(*
SPDX-FileCopyrightText: © 2026 Oleksandr Tiutyk <trofimich@gmail.com>
SPDX-License-Identifier: MIT
License: https://opensource.org/license/mit
*)

(*!
<summary>Provides lexical checks for directory and file path strings.</summary>
<description>
These checks perform no filesystem I/O, normalization or access checks. Passing does not certify acceptance by
a native service or target filesystem. The current filter is not a complete Windows, UNC or platform-specific
path validator; it does not validate reserved names or dot components. Callers must separately satisfy the
path requirements of the actual operation and target.
</description>
*)

{attribute 'no_explicit_call' := 'do not call this function block directly'}
PROGRAM PathHelper
VAR CONSTANT
	//! <summary>Drive-letter, colon and separator occupy the first three bytes of an absolute drive prefix.</summary>
	_DrivePrefixLength : UDINT := 3;
	//! <summary>Zero-based index of the colon immediately following a drive letter.</summary>
	_DriveColonIndex : UDINT := 1;
	//! <summary>Zero-based index of the separator following the drive colon.</summary>
	_DriveSeparatorIndex : UDINT := 2;
	//! <summary>Last index allowed in the initial separator pair before repeated separators are rejected.</summary>
	_LeadingSeparatorPairLastIndex : UDINT := 1;
END_VAR
VAR
	{attribute 'hide'} 
	_ClassName : STRING := __POUNAME();
END_VAR

//! <summary>Borrows the concrete class name for the lifetime of this instance; callers must not modify it.</summary>
{attribute 'monitoring' := 'call'}
PROPERTY ClassName : REFERENCE TO STRING
GET
ClassName REF= _ClassName;
END_GET
END_PROPERTY

(*!
<summary>Checks the lexical form of a directory path without accessing the filesystem.</summary>
<description>
Rejects an empty path, bytes below ASCII space, characters from the current forbidden set and repeated
slash/backslash separators beyond the leading pair. A colon is accepted only immediately after an ASCII drive
letter and before a separator. Relative paths and a trailing separator are not rejected solely for being
relative or trailing. Leading separator pairs are permitted lexically, but UNC server/share structure is not
checked and native network-path support is not implied. Reserved names, dot components and trailing
dots/spaces are not validated. TRUE means only that this filter passed; errorMessage is meaningful on FALSE.
Input is borrowed only for the call.
</description>
<param name="directoryPath">Directory path to inspect without modifying or retaining it.</param>
<param name="errorMessage">Reason for the first rejected condition.</param>
*)
METHOD IsValidDirectoryPath : BOOL
VAR_IN_OUT CONSTANT
	directoryPath : Tc2_System.T_MaxString;
END_VAR
VAR_OUTPUT
	errorMessage : WSTRING(255);
END_VAR
VAR
	i, j : UDINT;
	stringLength : UDINT;
	character : BYTE;

	(* Current lexical exclusions, not an OS-wide list. Caret is an existing library restriction;
	   the drive-letter exception below handles the only accepted colon position. *)
	invalidChars : STRING(8) := '<>"|?*^:';
END_VAR
stringLength := TOF_Core.Strings.GetLength(value := directoryPath);

IF stringLength = TOF_Core.UnsignedInt32.ZERO THEN
	errorMessage := "Path is empty";
	RETURN;
END_IF

FOR i := 0 TO stringLength - 1 DO
	character := directoryPath[i];

	(* A colon is allowed only in an absolute ASCII drive prefix. *)
	IF i = _DriveColonIndex AND_THEN character = Tc2_System.F_ToASC(str := ':') THEN

		IF stringLength >= _DrivePrefixLength
			AND_THEN (
				directoryPath[_DriveSeparatorIndex] = Tc2_System.F_ToASC(str := '\')
				OR_ELSE directoryPath[_DriveSeparatorIndex] = Tc2_System.F_ToASC(str := '/')
			)
			AND_THEN (
				(directoryPath[0] >= Tc2_System.F_ToASC(str := 'A')
					AND_THEN directoryPath[0] <= Tc2_System.F_ToASC(str := 'Z'))
				OR_ELSE (directoryPath[0] >= Tc2_System.F_ToASC(str := 'a')
					AND_THEN directoryPath[0] <= Tc2_System.F_ToASC(str := 'z'))
			)
		THEN
			CONTINUE;
		END_IF

	END_IF

	FOR j := 0 TO TOF_Core.Strings.GetLength(value := invalidChars) - 1 DO

		IF character = invalidChars[j] THEN
			errorMessage := TOF_Core.WideStrings.Concat255(
				"The forbidden character '",
				TO_WSTRING(Tc2_System.F_ToCHR(c := character)),
				"' at position ",
				TO_WSTRING(i + 1)
			);
			RETURN;
		END_IF

	END_FOR

	IF character < TOF_Core.Strings.ASCII_SPACE THEN
		errorMessage := TOF_Core.WideStrings.Concat255(
			"The forbidden character with code ",
			TO_WSTRING(character),
			" at position ",
			TO_WSTRING(i + 1)
		);
		RETURN;
	END_IF

	IF i > _LeadingSeparatorPairLastIndex
		AND_THEN (character = Tc2_System.F_ToASC(str := '\') OR_ELSE character = Tc2_System.F_ToASC(str := '/'))
		AND_THEN (
			directoryPath[i - 1] = Tc2_System.F_ToASC(str := '\')
			OR_ELSE directoryPath[i - 1] = Tc2_System.F_ToASC(str := '/')
		)
	THEN
		errorMessage := TOF_Core.WideStrings.Concat255("Several slashes one by one at position ", TO_WSTRING(i + 1));
		RETURN;
	END_IF

END_FOR

IsValidDirectoryPath := TRUE;
END_METHOD

(*!
<summary>Checks the lexical form of a file path and rejects a trailing separator.</summary>
<description>
Borrows the path only for this call. Returns FALSE with errorMessage for an empty path, a forbidden character,
repeated separators beyond the leading pair, or a final slash or backslash. A drive-letter colon is allowed
only before a slash or backslash. TRUE means the lexical checks passed; it does not establish file existence,
access rights or acceptance by the target filesystem. No filesystem I/O is performed. Relative paths are not
rejected solely for being relative. Leading separator pairs do not establish a valid UNC path; reserved names,
dot components and trailing dots/spaces are not validated. errorMessage is meaningful only when FALSE is
returned.
</description>
<param name="filePath">File path to inspect without modifying or retaining it.</param>
<param name="errorMessage">Receives the reason for the first rejected condition.</param>
*)
METHOD IsValidFilePath : BOOL
VAR_IN_OUT CONSTANT
	filePath : Tc2_System.T_MaxString;
END_VAR
VAR_OUTPUT
	errorMessage : WSTRING(255);
END_VAR
VAR
	i, j : UDINT;
	stringLength : UDINT;
	character : BYTE;

	(* Current lexical exclusions, not an OS-wide list. Caret is an existing library restriction;
	   the drive-letter exception below handles the only accepted colon position. *)
	invalidChars : STRING(8) := '<>"|?*^:';
END_VAR
stringLength := TOF_Core.Strings.GetLength(value := filePath);

IF stringLength = TOF_Core.UnsignedInt32.ZERO THEN
	errorMessage := "Path is empty";
	RETURN;
END_IF

FOR i := 0 TO stringLength - 1 DO
	character := filePath[i];

	(* A colon is allowed only in an absolute ASCII drive prefix. *)
	IF i = _DriveColonIndex AND_THEN character = Tc2_System.F_ToASC(str := ':') THEN

		IF stringLength >= _DrivePrefixLength
			AND_THEN (
				filePath[_DriveSeparatorIndex] = Tc2_System.F_ToASC(str := '\')
				OR_ELSE filePath[_DriveSeparatorIndex] = Tc2_System.F_ToASC(str := '/')
			)
			AND_THEN (
				(filePath[0] >= Tc2_System.F_ToASC(str := 'A')
					AND_THEN filePath[0] <= Tc2_System.F_ToASC(str := 'Z'))
				OR_ELSE (filePath[0] >= Tc2_System.F_ToASC(str := 'a')
					AND_THEN filePath[0] <= Tc2_System.F_ToASC(str := 'z'))
			)
		THEN
			CONTINUE;
		END_IF

	END_IF

	FOR j := 0 TO TOF_Core.Strings.GetLength(value := invalidChars) - 1 DO

		IF character = invalidChars[j] THEN
			errorMessage := TOF_Core.WideStrings.Concat255(
				"The forbidden character '",
				TO_WSTRING(Tc2_System.F_ToCHR(c := character)),
				"' at position ",
				TO_WSTRING(i + 1)
			);
			RETURN;
		END_IF

	END_FOR

	IF character < TOF_Core.Strings.ASCII_SPACE THEN
		errorMessage := TOF_Core.WideStrings.Concat255(
			"The forbidden character with code ",
			TO_WSTRING(character),
			" at position ",
			TO_WSTRING(i + 1)
		);
		RETURN;
	END_IF

	IF i > _LeadingSeparatorPairLastIndex
		AND_THEN (character = Tc2_System.F_ToASC(str := '\') OR_ELSE character = Tc2_System.F_ToASC(str := '/'))
		AND_THEN (
			filePath[i - 1] = Tc2_System.F_ToASC(str := '\')
			OR_ELSE filePath[i - 1] = Tc2_System.F_ToASC(str := '/')
		)
	THEN
		errorMessage := TOF_Core.WideStrings.Concat255("Several slashes one by one at position ", TO_WSTRING(i + 1));
		RETURN;
	END_IF

	IF i = stringLength - 1
		AND_THEN (character = Tc2_System.F_ToASC(str := '\') OR_ELSE character = Tc2_System.F_ToASC(str := '/'))
	THEN
		errorMessage := "Slash at the end of the path";
		RETURN;
	END_IF

END_FOR

IsValidFilePath := TRUE;
END_METHOD

//! <summary>Borrows the compiler-initialized namespace; callers must not modify the returned reference.</summary>
{attribute 'monitoring' := 'call'}
PROPERTY NamespaceName : REFERENCE TO STRING
GET
NamespaceName REF= CurrentNamespace.Name;
END_GET
END_PROPERTY

END_PROGRAM

(* stored: Version 1.1.0.1
   POU PathHelper: Id {0dca2365-65a2-482c-a73e-d706575b93b9}, SpecialFunc None
   Property ClassName: Id {bcad59d0-30a2-4095-8b10-42c3bd512232}
   Get Get: Id {4ebc6fc7-9213-424f-b2ff-4e572f38dc62}
   Method IsValidDirectoryPath: Id {74a38896-f3ee-456c-865c-7f0b909dbd4e}
   Method IsValidFilePath: Id {c79d4e63-0f05-42ae-918f-7c9d81a28bdc}
   Property NamespaceName: Id {03b769a2-dbc8-4792-82dc-d2506f34e5a7}
   Get Get: Id {d7e4e13f-8a4a-4bb5-a58d-6cd9c5969c93} *)
